// SIMATIC S7-200 project (STEP 7-Micro/WIN), CPU 224 REL 02.01

SYMBOL_TABLE USER1
start            I0.0     // start
stopp            I0.1     // stop
s1               I0.2     // cb tren
s2               I0.3     // cb duoi
s3               I0.4     // cb nguoi
xuong            Q0.0     // di xuong
len              Q0.1     // di len
END_SYMBOL_TABLE

ORGANIZATION_BLOCK MAIN:OB1
TITLE=PROGRAM COMMENTS
BEGIN
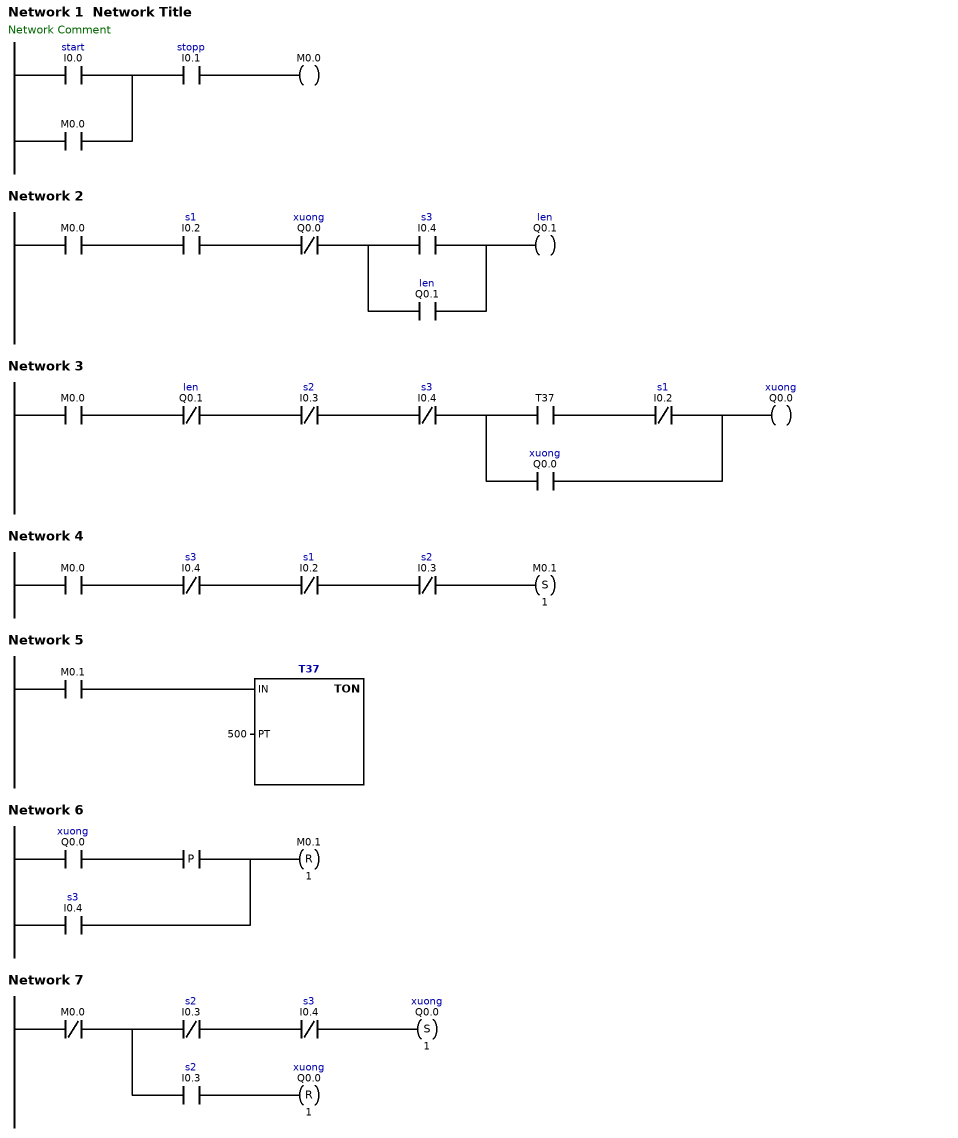
Network 1 // Network Title
// Network Comment
LD     start:I0.0
O      M0.0
A      stopp:I0.1
=      M0.0
Network 2
LD     M0.0
A      s1:I0.2
AN     xuong:Q0.0
LD     s3:I0.4
O      len:Q0.1
ALD
=      len:Q0.1
Network 3
LD     M0.0
AN     len:Q0.1
AN     s2:I0.3
AN     s3:I0.4
LD     T37
AN     s1:I0.2
O      xuong:Q0.0
ALD
=      xuong:Q0.0
Network 4
LD     M0.0
AN     s3:I0.4
AN     s1:I0.2
AN     s2:I0.3
S      M0.1, 1
Network 5
LD     M0.1
TON    T37, 500
Network 6
LD     xuong:Q0.0
EU
O      s3:I0.4
R      M0.1, 1
Network 7
LDN    M0.0
LPS
AN     s2:I0.3
AN     s3:I0.4
S      xuong:Q0.0, 1
LPP
A      s2:I0.3
R      xuong:Q0.0, 1
END_ORGANIZATION_BLOCK
